// TwinCAT 3 PLC project Plc1
// ProgramVersion: 3.1.4023.0
// libraries:
//   Tc2_Standard, * (Beckhoff Automation GmbH)
//   Tc2_System, * (Beckhoff Automation GmbH)
//   Tc3_Module, * (Beckhoff Automation GmbH)
// project tree:
//   DUTs/ E_Colors.TcDUT
//   / PlcTask.TcTTO
//   POUs/ FB_Color.TcPOU, MAIN.TcPOU
// real-time tasks:
//   TASK PlcTask: cycle T#10ms, priority 20, ADS port 350

CONFIGURATION Plc1
    RESOURCE PLC ON TwinCAT3
        TASK PlcTask(INTERVAL := T#10ms, PRIORITY := 20);
        PROGRAM MAIN WITH PlcTask : MAIN;
    END_RESOURCE
END_CONFIGURATION

// ---- DUTs/E_Colors.TcDUT
{attribute 'qualified_only'}
{attribute 'strict'}
TYPE E_Colors :
(
	red,
	orange,
	yellow,
	green,
	blue
);
END_TYPE

// ---- POUs/MAIN.TcPOU
PROGRAM MAIN
VAR
	fbColor	: FB_Color;
END_VAR

END_PROGRAM

// ---- POUs/FB_Color.TcPOU
FUNCTION_BLOCK FB_Color
VAR_INPUT
END_VAR
VAR_OUTPUT
END_VAR
VAR
END_VAR

END_FUNCTION_BLOCK
